(* Logix 5000 project; controller RSL5k_18_Template_noLib Emulate 5570 rev 32.11; software revision 32.02; part 5 of 16 *)
(* tags used below, declared in another part *)
   Inp_Hand : BOOL;   // 1=Acquire Hand (typ. hardwired local), 0=Release Hand
   Inp_Ovrd : BOOL;   // 1=Acquire Override (higher priority program logic), 0=Release Override
   Inp_ExtInh : BOOL;   // 1=Inhibit External Acquisition, 0=Allow External Acquisition
   Cfg_HasOper : BOOL;   // 1=Operator (unlocked) exists, can be selected
   Cfg_HasOperLocked : BOOL;   // 1=Operator Locked exists, can be selected
   Cfg_HasProg : BOOL;   // 1=Program (unlocked) exists, can be selected
   Cfg_HasProgLocked : BOOL;   // 1=Program Locked exists, can be selected
   Cfg_HasExt : BOOL;   // 1=External exists, can be selected
   Cfg_HasMaint : BOOL;   // 1=Maintenance exists, can be selected
   Cfg_HasMOoS : BOOL;   // 1=Maintenance Out of Service exists, can be selected
   Cfg_OvrdOverLock : BOOL;   // 1=Override supersedes Prog/Oper Lock, 0=don't override Lock
   Cfg_ExtOverLock : BOOL;   // 1=External supersedes Prog/Oper Lock, 0=don't override Lock
   Cfg_ProgNormal : BOOL;   // Normal Source: 1=Program if no requests; 0=Operator if no requests
   Cfg_PCmdPriority : BOOL;   // Command Priority: 1=Program Cmds Win; 0=Operator Cmds Win
   Cfg_PCmdProgAsLevel : BOOL;   // 1=PCmd_Prog used as a Level (1=Prog, 0=Oper)
   Cfg_PCmdLockAsLevel : BOOL;   // 1=PCmd_Lock used as a Level (1=Lock, 0=Unlock)
   Cfg_ExtAcqAsLevel : BOOL;   // 1=XCmd_Acq used as Level (1=Acq, 0=Rel)
   PCmd_Prog : BOOL;   // Program Command to select Program (Oper to Prog)
   PCmd_Lock : BOOL;   // Program Command to Lock Program (disallow Operator)
   MCmd_Acq : BOOL;   // Maintenance Command to Acquire (Oper/Prog/Ovrd to Maint)
   XCmd_Acq : BOOL;   // External Command to Acquire
   XCmd_Rel : BOOL;   // External Command to Release
   OCmd_Lock : BOOL;   // Operator Command to Lock Operator (disallow Program)
   Sts_eSrc : INT;   // Selection enum: .8=Ext, .7=OoS, .6=Oper, .5=Prog, .4=Ovrd, .3=Maint, .2=Hand, .1=Norm, .0=Lock
   Sts_bSrc : INT;   // Active Selection bitmap (for HMI totem pole)
   Sts_Hand : BOOL;   // 1=Hand is selected (supersedes OoS, Maint, Ovrd, Ext, Prog, Oper)
   Sts_OoS : BOOL;   // 1=Out of Service is selected (supersedes Maint, Ovrd, Ext, Prog, Oper)
   Sts_Maint : BOOL;   // 1=Maintenance is selected (supersedes Ovrd, Ext, Prog, Oper)
   Sts_Ovrd : BOOL;   // 1=Override is selected (supersedes Ext, Prog, Oper)
   Sts_Ext : BOOL;   // 1=External is selected (supersedes Prog, Oper)
   Sts_Prog : BOOL;   // 1=Program is selected
   Sts_ProgLocked : BOOL;   // 1=Program is selected and Locked
   Sts_Oper : BOOL;   // 1=Operator is selected
   Sts_OperLocked : BOOL;   // 1=Operator is selected and Locked
   Sts_ProgOperSel : BOOL;   // Prog/Oper selection (latch) state, 1=Program, 0=Operator
   Sts_ProgOperLock : BOOL;   // Prog/Oper lock (latch) state, 1=Locked, 0=Unlocked
   Sts_Normal : BOOL;   // 1=Selection equals the Normal (Prog or Oper)
   Sts_ProgReqInh : BOOL;   // 1=Program request inhibited, cannot Get to Program from Current State
   Sts_ExtReqInh : BOOL;   // 1=External request inhibited
   Sts_MAcqRcvd : BOOL;   // 1=Maintenance Acquire command received this scan
   MRdy_OoS : BOOL;   // 1=Ready for MCmd_OoS (enables HMI button)
   MRdy_IS : BOOL;   // 1=Ready for MCmd_IS (enables HMI button)
   MRdy_Acq : BOOL;   // 1=Ready for MCmd_Acq (enables HMI button)
   MRdy_Rel : BOOL;   // 1=Ready for MCmd_Rel (enables HMI button)
   XRdy_Acq : BOOL;   // 1=Ready for XCmd_Acq (enables HMI button)
   XRdy_Rel : BOOL;   // 1=Ready for XCmd_Rel (enables HMI button)
   ORdy_Oper : BOOL;   // 1=Ready for OCmd_Oper (enables HMI button)
   ORdy_Prog : BOOL;   // 1=Ready for OCmd_Prog (enables HMI button)
   ORdy_Lock : BOOL;   // 1=Ready for OCmd_Lock (enables HMI button)
   ORdy_Unlock : BOOL;   // 1=Ready for OCmd_Unlock (enables HMI button)
   ORdy_Normal : BOOL;   // 1=Ready for OCmd_Normal (enables HMI button)
   P_CmdSrc : BOOL;   // Unique Parameter Name for auto - discovery
   Wrk_ProgOperSel : BOOL;   // Internal Program (1) / Operator (0) selection result
   Wrk_ProgOperLock : BOOL;   // Internal Prog/Oper Lock (1) / Unlock (0) selection result
   Wrk_Prog : BOOL;   // Internal Program (1) / Operator (0) selection progress
   Wrk_MOoS : BOOL;   // Internal Maintenance Out of Service (1) / In Service (0) latch
   Wrk_Maint : BOOL;   // Internal Maintenance Acquire (1) / Release (0) latch
   Wrk_Lock : BOOL;   // Internal Prog/Oper Lock (1) / Unlock (0) selection progress
   Wrk_Init : BOOL;   // 1=Initialized, 0=Initialization is required (e.g., powerup)
   Wrk_Ext : BOOL;   // Internal latch of External selection (1=Ext acquired)
(* P_CmdSrc, continued *)

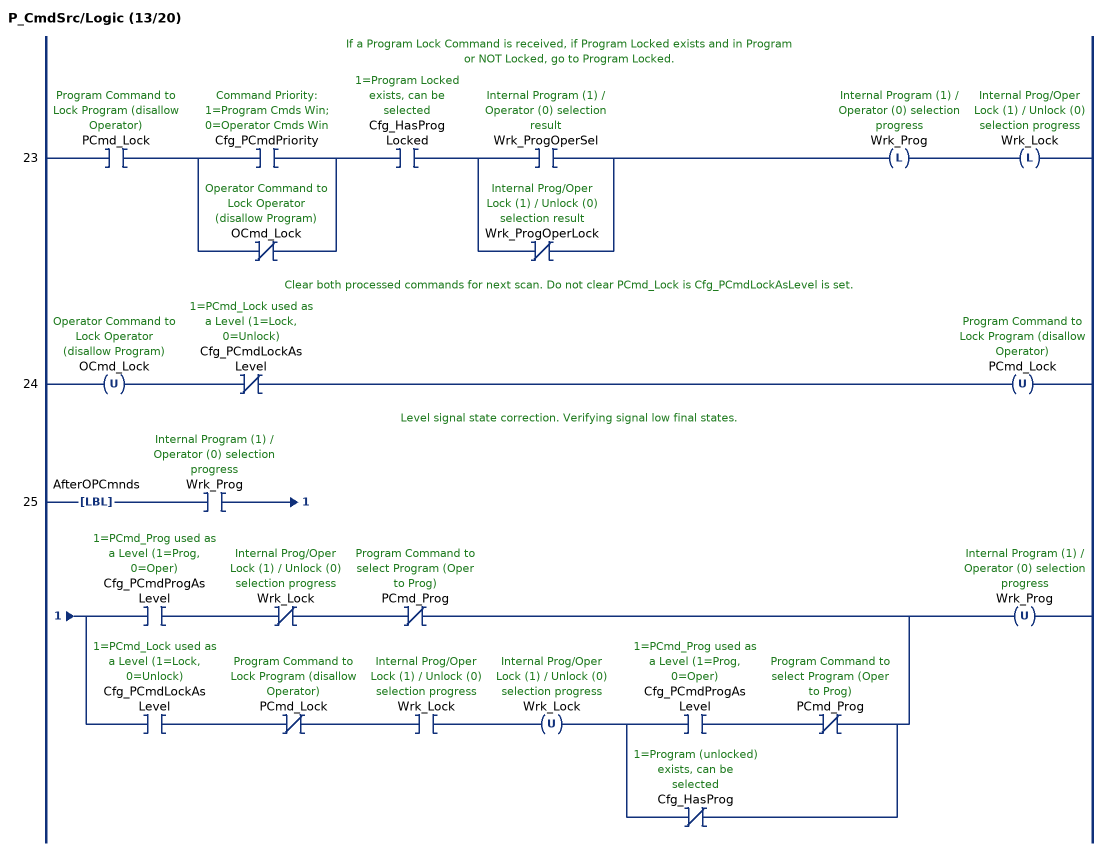
   // If a Program Lock Command is received, if Program Locked exists and in Program
   // or NOT Locked, go to Program Locked.
   23: XIC(PCmd_Lock)[XIC(Cfg_PCmdPriority) ,XIO(OCmd_Lock) ]XIC(Cfg_HasProgLocked)[XIC(Wrk_ProgOperSel) ,XIO(Wrk_ProgOperLock) ]OTL(Wrk_Prog)OTL(Wrk_Lock);
   // Clear both processed commands for next scan. Do not clear PCmd_Lock is Cfg_PCmdLockAsLevel is set.
   24: OTU(OCmd_Lock)XIO(Cfg_PCmdLockAsLevel)OTU(PCmd_Lock);
   // Level signal state correction. Verifying signal low final states.
   25: LBL(AfterOPCmnds)XIC(Wrk_Prog)[XIC(Cfg_PCmdProgAsLevel) XIO(Wrk_Lock) XIO(PCmd_Prog) ,XIC(Cfg_PCmdLockAsLevel) XIO(PCmd_Lock) XIC(Wrk_Lock) OTU(Wrk_Lock) [XIC(Cfg_PCmdProgAsLevel) XIO(PCmd_Prog) ,XIO(Cfg_HasProg) ] ]OTU(Wrk_Prog);
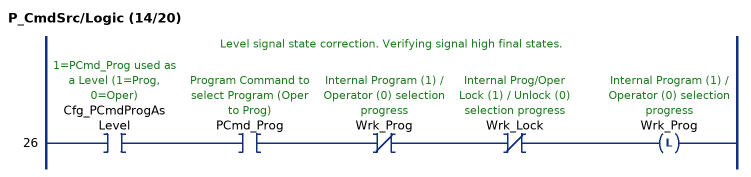
   // Level signal state correction. Verifying signal high final states.
   26: XIC(Cfg_PCmdProgAsLevel)XIC(PCmd_Prog)XIO(Wrk_Prog)XIO(Wrk_Lock)OTL(Wrk_Prog);
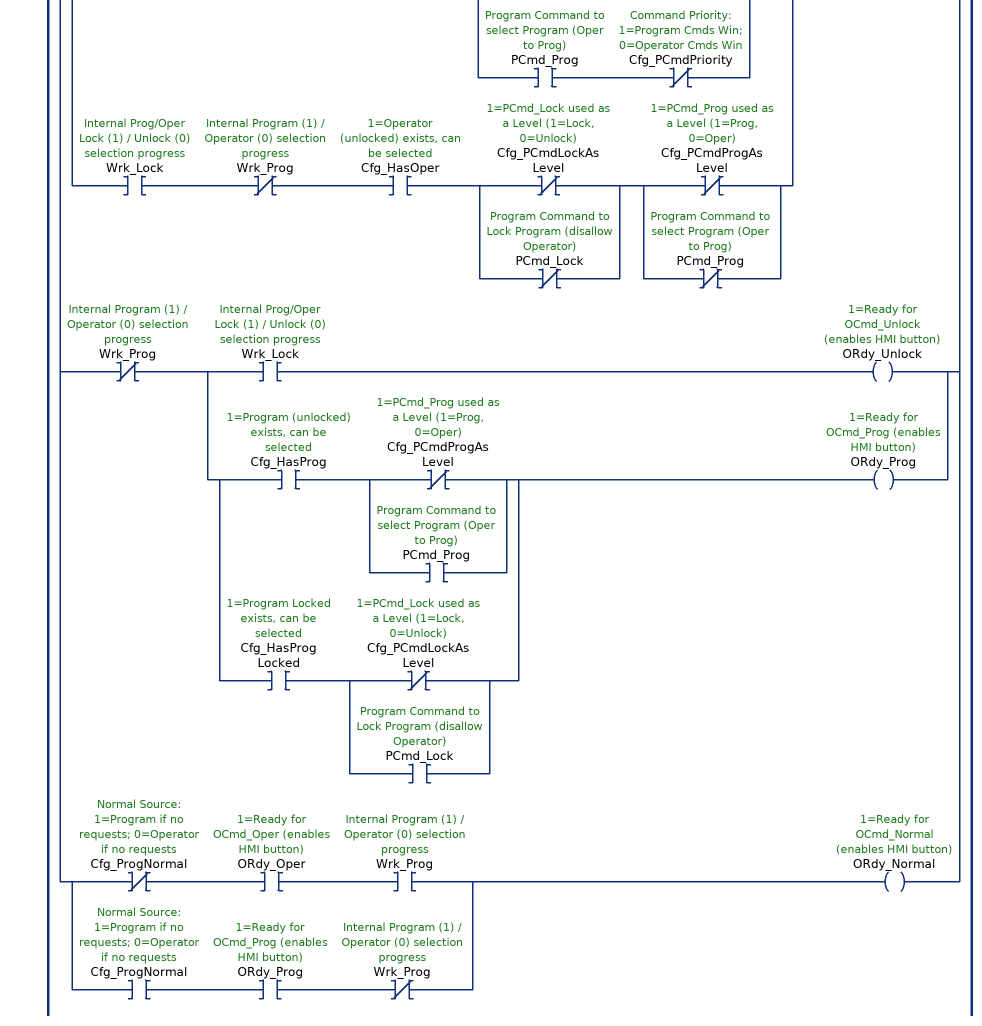
   // ============================================================
   // MAINTENANCE AND OPERATOR COMMAND READIES
   // ============================================================
   // This rung generates the "ORdy_" and "MRdy_" bits that signify to the
   // HMI that the corresponding command should "do" something
   // and the command button should be enabled on the display.
   // NOTE ON MAINTENANCE ACQUIRE: Ready for MCmd_Acq if Maintenance
   // is allowed and the internal Maintenance latch is NOT set.  However,
   // we need to display Ready even if latch IS set so that Sts_MAcqRcvd
   // can blink to reset an external Maintenance expiration timer!!!
   // #####  V4.10.00  2019-03-08:  Added XRdy_Acq, XRdy_Rel so External Acq/Rel can be used on HMI .  #####
   27: [XIC(Cfg_HasMaint) [OTE(MRdy_Acq) ,XIC(Wrk_Maint) OTE(MRdy_Rel) ] ,XIC(Cfg_HasMOoS) [XIC(Wrk_MOoS) OTE(MRdy_IS) ,XIO(Wrk_MOoS) OTE(MRdy_OoS) ] ,XIC(Cfg_HasExt) XIO(Cfg_ExtAcqAsLevel) [XIC(Wrk_Ext) OTE(XRdy_Rel) ,XIO(Wrk_Ext) XIO(Inp_ExtInh) OTE(XRdy_Acq) ] ,XIO(Wrk_Lock) XIC(Cfg_HasOperLocked) OTE(ORdy_Lock) ,[XIO(Wrk_Lock) XIC(Wrk_Prog) [XIC(Cfg_HasOper) XIO(Cfg_PCmdProgAsLevel) ,XIC(Cfg_HasOperLocked) [XIO(Cfg_PCmdProgAsLevel) ,XIC(PCmd_Prog) XIO(Cfg_PCmdPriority) ] ] ,XIC(Wrk_Lock) XIO(Wrk_Prog) XIC(Cfg_HasOper) [XIO(Cfg_PCmdLockAsLevel) ,XIO(PCmd_Lock) ] [XIO(Cfg_PCmdProgAsLevel) ,XIO(PCmd_Prog) ] ] OTE(ORdy_Oper) ,XIO(Wrk_Prog) [XIC(Wrk_Lock) OTE(ORdy_Unlock) ,[XIC(Cfg_HasProg) [XIO(Cfg_PCmdProgAsLevel) ,XIC(PCmd_Prog) ] ,XIC(Cfg_HasProgLocked) [XIO(Cfg_PCmdLockAsLevel) ,XIC(PCmd_Lock) ] ] OTE(ORdy_Prog) ] ,[XIO(Cfg_ProgNormal) XIC(ORdy_Oper) XIC(Wrk_Prog) ,XIC(Cfg_ProgNormal) XIC(ORdy_Prog) XIO(Wrk_Prog) ] OTE(ORdy_Normal) ];
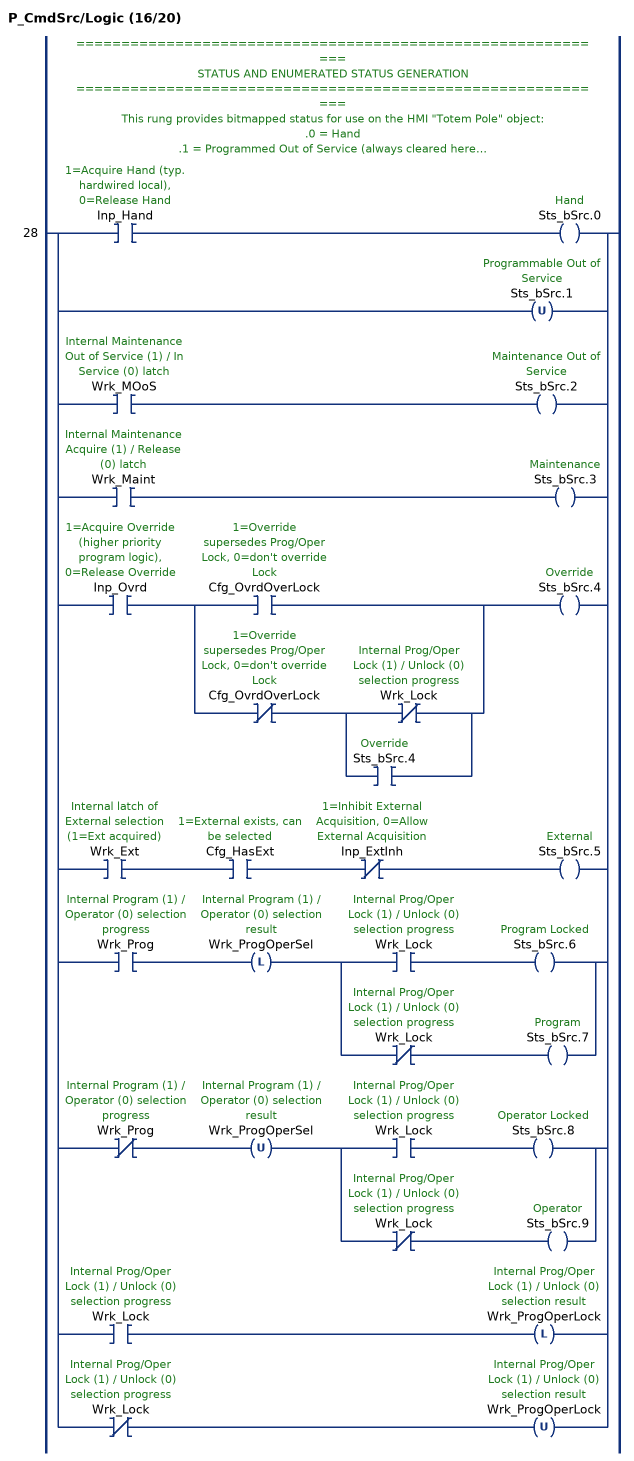
   // ============================================================
   // STATUS AND ENUMERATED STATUS GENERATION
   // ============================================================
   // This rung provides bitmapped status for use on the HMI "Totem Pole" object:
   // .0 = Hand
   // .1 = Programmed Out of Service (always cleared here)
   // .2 = Maintenance Out of Service
   // .3 = Maintenance
   // .4= Override
   // .5 = External
   // .6 = Program Locked
   // .7 = Program
   // .8 = Operator Locked
   // .9 = Operator
   // In addition, the final selections of the Program / Operator selection latch
   // and the Prog/Oper lock latch are captured for use next scan.
   // #####  V4.10.00  2019-03-08:  Added XCmd_Acq, XCmd_Rel, Cfg_ExtAcqAsLevel, removed Inp_Ext.  #####
   28: [XIC(Inp_Hand) OTE(Sts_bSrc.0) ,OTU(Sts_bSrc.1) ,XIC(Wrk_MOoS) OTE(Sts_bSrc.2) ,XIC(Wrk_Maint) OTE(Sts_bSrc.3) ,XIC(Inp_Ovrd) [XIC(Cfg_OvrdOverLock) ,XIO(Cfg_OvrdOverLock) [XIO(Wrk_Lock) ,XIC(Sts_bSrc.4) ] ] OTE(Sts_bSrc.4) ,XIC(Wrk_Ext) XIC(Cfg_HasExt) XIO(Inp_ExtInh) OTE(Sts_bSrc.5) ,XIC(Wrk_Prog) OTL(Wrk_ProgOperSel) [XIC(Wrk_Lock) OTE(Sts_bSrc.6) ,XIO(Wrk_Lock) OTE(Sts_bSrc.7) ] ,XIO(Wrk_Prog) OTU(Wrk_ProgOperSel) [XIC(Wrk_Lock) OTE(Sts_bSrc.8) ,XIO(Wrk_Lock) OTE(Sts_bSrc.9) ] ,XIC(Wrk_Lock) OTL(Wrk_ProgOperLock) ,XIO(Wrk_Lock) OTU(Wrk_ProgOperLock) ];
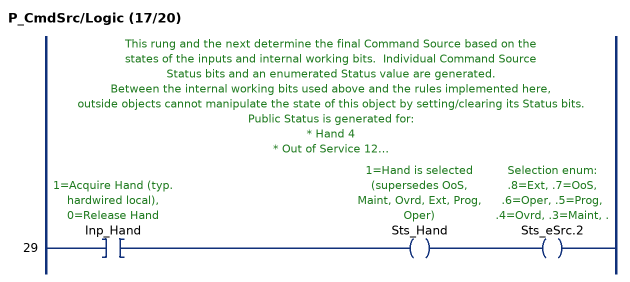
   // This rung and the next determine the final Command Source based on the
   // states of the inputs and internal working bits.  Individual Command Source
   // Status bits and an enumerated Status value are generated.
   // Between the internal working bits used above and the rules implemented here,
   // outside objects cannot manipulate the state of this object by setting/clearing its Status bits.
   // Public Status is generated for:
   // * Hand 4
   // * Out of Service 129
   // * Maintenance 8
   // * Override 16
   // * External 256
   // * Program 32
   // * Operator 64
   // * Program / Operator Lock status 33/65
   // * Command Source = Normal 34/66
   29: XIC(Inp_Hand)OTE(Sts_Hand)OTE(Sts_eSrc.2);
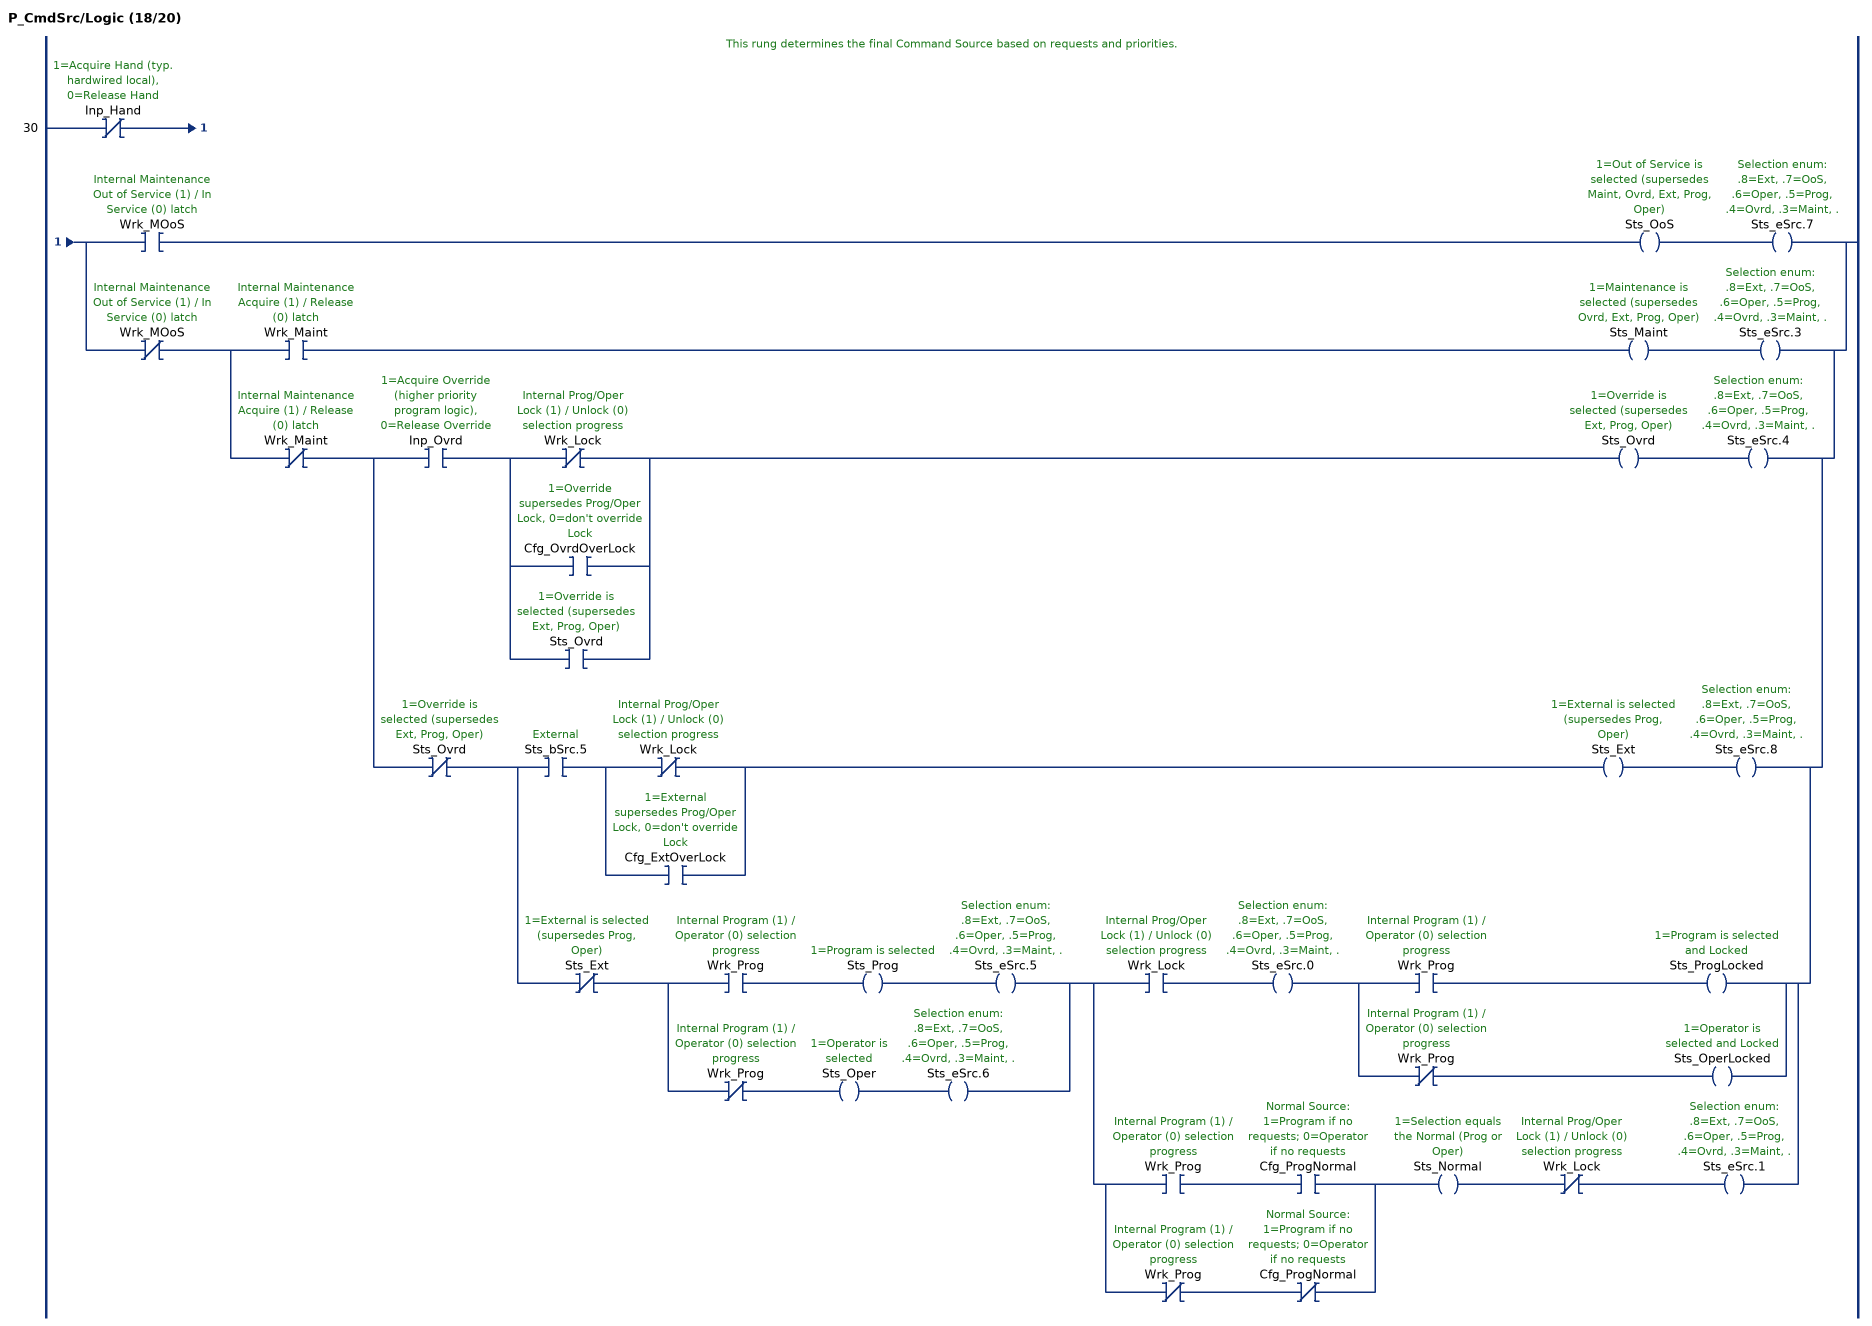
   // This rung determines the final Command Source based on requests and priorities.
   30: XIO(Inp_Hand)[XIC(Wrk_MOoS) OTE(Sts_OoS) OTE(Sts_eSrc.7) ,XIO(Wrk_MOoS) [XIC(Wrk_Maint) OTE(Sts_Maint) OTE(Sts_eSrc.3) ,XIO(Wrk_Maint) [XIC(Inp_Ovrd) [XIO(Wrk_Lock) ,XIC(Cfg_OvrdOverLock) ,XIC(Sts_Ovrd) ] OTE(Sts_Ovrd) OTE(Sts_eSrc.4) ,XIO(Sts_Ovrd) [XIC(Sts_bSrc.5) [XIO(Wrk_Lock) ,XIC(Cfg_ExtOverLock) ] OTE(Sts_Ext) OTE(Sts_eSrc.8) ,XIO(Sts_Ext) [XIC(Wrk_Prog) OTE(Sts_Prog) OTE(Sts_eSrc.5) ,XIO(Wrk_Prog) OTE(Sts_Oper) OTE(Sts_eSrc.6) ] [XIC(Wrk_Lock) OTE(Sts_eSrc.0) [XIC(Wrk_Prog) OTE(Sts_ProgLocked) ,XIO(Wrk_Prog) OTE(Sts_OperLocked) ] ,[XIC(Wrk_Prog) XIC(Cfg_ProgNormal) ,XIO(Wrk_Prog) XIO(Cfg_ProgNormal) ] OTE(Sts_Normal) XIO(Wrk_Lock) OTE(Sts_eSrc.1) ] ] ] ] ];
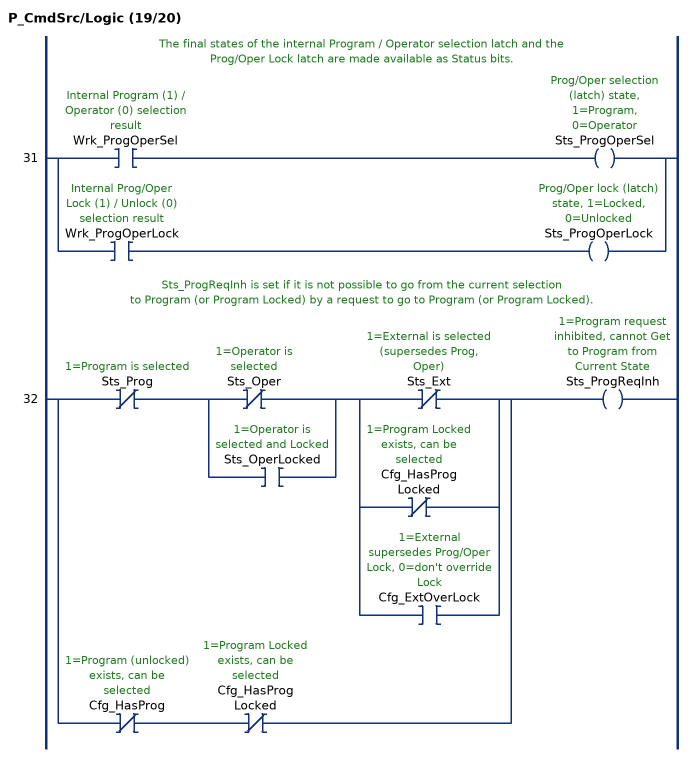
   // The final states of the internal Program / Operator selection latch and the
   // Prog/Oper Lock latch are made available as Status bits.
   31: [XIC(Wrk_ProgOperSel) OTE(Sts_ProgOperSel) ,XIC(Wrk_ProgOperLock) OTE(Sts_ProgOperLock) ];
   // Sts_ProgReqInh is set if it is not possible to go from the current selection
   // to Program (or Program Locked) by a request to go to Program (or Program Locked).
   32: [XIO(Sts_Prog) [XIO(Sts_Oper) ,XIC(Sts_OperLocked) ] [XIO(Sts_Ext) ,XIO(Cfg_HasProgLocked) ,XIC(Cfg_ExtOverLock) ] ,XIO(Cfg_HasProg) XIO(Cfg_HasProgLocked) ]OTE(Sts_ProgReqInh);
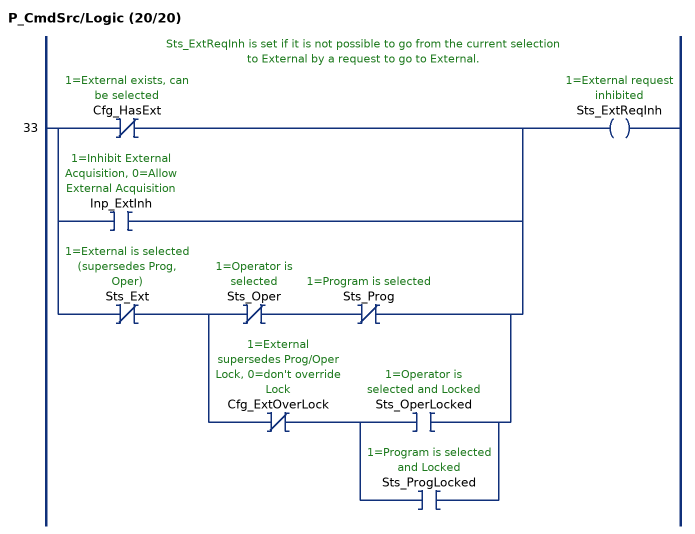
   // Sts_ExtReqInh is set if it is not possible to go from the current selection
   // to External by a request to go to External.
   33: [XIO(Cfg_HasExt) ,XIC(Inp_ExtInh) ,XIO(Sts_Ext) [XIO(Sts_Oper) XIO(Sts_Prog) ,XIO(Cfg_ExtOverLock) [XIC(Sts_OperLocked) ,XIC(Sts_ProgLocked) ] ] ]OTE(Sts_ExtReqInh);
END_ROUTINE

ROUTINE Prescan   (* ladder *)
// Sets internal state and enumerated / bit status to "not initialized".
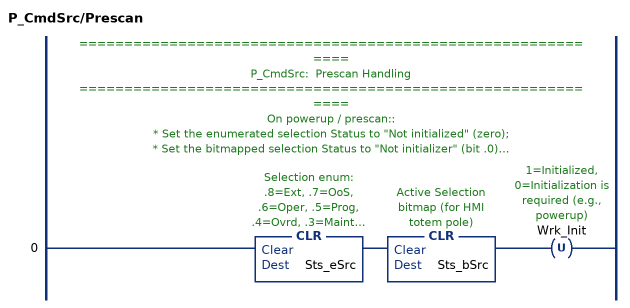
   // ============================================================
   // P_CmdSrc:  Prescan Handling
   // ============================================================
   // On powerup / prescan::
   // * Set the enumerated selection Status to "Not initialized" (zero);
   // * Set the bitmapped selection Status to "Not initializer" (bit .0);
   // * Flag the instruction to execute the initialization rungs when run.
   0: CLR(Sts_eSrc)CLR(Sts_bSrc)OTU(Wrk_Init);
END_ROUTINE
END_ADD_ON_INSTRUCTION

ADD_ON_INSTRUCTION P_Gate   (* revision 4.10 .00 Release, vendor Rockwell Automation, ExecutePrescan, ExecuteEnableInFalse *)
// Condition Gate/Delay
// Revision note:
// See Instruction Help for a summary of changes, and see 4.10 Release Notes for details.
// Help:
// Copyright © Rockwell Automation, Inc.  All Rights Reserved.
// This Instruction provides a "gate" for a discrete Input signal and
// provides on-delay and off-delay timing for the gated signal.
// When the Gate input is true, the instruction Input is passed through
// to the Output, with on-delay and off-delay timing applied.
// When the Gate input is false, the Output is kept off
// (note: off-delay still applies!)
// This instruction is usually used between a comparison
// (analog threshold with deadband or discrete logic)
// and a P_Alarm instance, but may be used as a
// gated on-delay/off-delay timer generally.
// When EnableIn  is FALSE (e.g., on a false LD rung), the Input "Inp"
// is inverted.  Note that the Gate input (Inp_Gate) is NOT inverted!!!
// SUMMARY OF CHANGES FROM PREVIOUS VERSION (4.00.00)
// See 4.10 Release Notes for details.
// * Unmodified, up-rev only for Library 4.10.00
// SUMMARY OF CHANGES FROM PREVIOUS VERSION (3.5-01)
// See 4.00 Release Notes for details.
// * Changed Inf_ items to HMI_ (e.g., HMI_Lib, HMI_Type).
// * Changed delay time configuration items to REAL seconds
VAR_INPUT
   Inp : BOOL; {visible}   // Input Condition: e.g., result of comparison
   Inp_Gate : BOOL := 1; {visible}   // Gate Input: 1=enable On Delay / Off Delay after Gate Delay, 0=disable
   Cfg_GateDly : REAL;   // Gate Delay (s): time after Gate Input true to enable On/Off Delay
   Cfg_OnDly : REAL;   // On Delay (s): If Gate Delay done, time Inp must be true to set Out true
   Cfg_OffDly : REAL;   // Off Delay (s): Time after Inp or Gate goes to 0 for Out to go to 0
END_VAR
VAR_OUTPUT
   Out : BOOL; {access Read Only, visible}   // Output after On Delay, Off Delay, enabled by Gate
   Sts_Gate : BOOL; {access Read Only, visible}   // 1=Gate Delay done, Output is enabled
   Sts_Err : BOOL; {access Read Only, visible}   // 1=Error in Config (see detail Err_ bits for reason), display icon
   Err_Timer : BOOL; {access Read Only}   // 1=Error in Config: On Delay, Off Delay, Gate Delay Time Invalid (use 0 to 2147483 s)
   P_Gate : BOOL;   // Unique Parameter Name for auto - discovery
END_VAR
VAR
   Wrk_OffDlyT : TIMER; {access Read Only}   // Off Delay Timer
   Wrk_OnDlyT : TIMER; {access Read Only}   // On Delay Timer
   Wrk_GateT : TIMER; {access Read Only}   // Gate Delay Timer
   Cfg_InpCond : STRING_20 := 'Input Condition';   // Displayed text of P_Gate's Input (Inp) Condition
   HMI_Lib : STRING_12 := 'RA-BAS'; {access Read Only}   // Display Library for Faceplate call-up
   HMI_Type : STRING_16 := 'P_Gate'; {access Read Only}   // Must contain AOI name, used for HMI and Information S/W
   Cfg_GateCond : STRING_20 := 'Gating Condition';   // Displayed text of P_Gate's Gating (Inp_Gate) Condition
   HMI_Tab : SINT;   // Tab to display (FTView ME)
END_VAR

ROUTINE EnableInFalse   (* ladder *)
// Same as main Logic routine, except Inp is inverted (for use in LD logic)  (Inp_Gate is NOT inverted!!!)
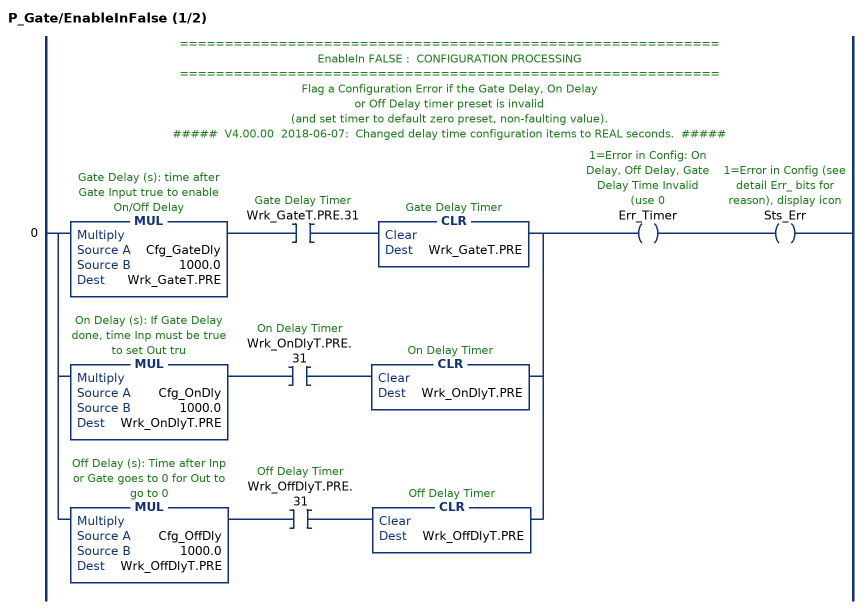
   // ============================================================
   // EnableIn FALSE :  CONFIGURATION PROCESSING
   // ============================================================
   // Flag a Configuration Error if the Gate Delay, On Delay
   // or Off Delay timer preset is invalid
   // (and set timer to default zero preset, non-faulting value).
   // #####  V4.00.00  2018-06-07:  Changed delay time configuration items to REAL seconds.  #####
   0: [MUL(Cfg_GateDly,1000.0,Wrk_GateT.PRE) XIC(Wrk_GateT.PRE.31) CLR(Wrk_GateT.PRE) ,MUL(Cfg_OnDly,1000.0,Wrk_OnDlyT.PRE) XIC(Wrk_OnDlyT.PRE.31) CLR(Wrk_OnDlyT.PRE) ,MUL(Cfg_OffDly,1000.0,Wrk_OffDlyT.PRE) XIC(Wrk_OffDlyT.PRE.31) CLR(Wrk_OffDlyT.PRE) ]OTE(Err_Timer)OTE(Sts_Err);
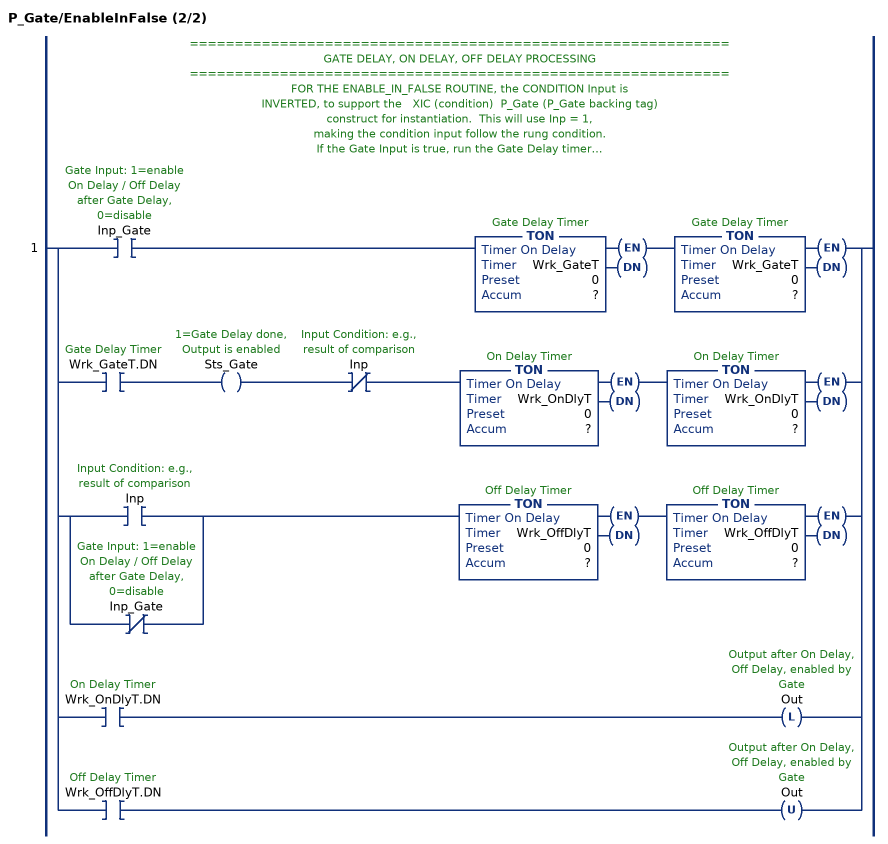
   // ============================================================
   // GATE DELAY, ON DELAY, OFF DELAY PROCESSING
   // ============================================================
   // FOR THE ENABLE_IN_FALSE ROUTINE, the CONDITION Input is
   // INVERTED, to support the   XIC (condition)  P_Gate (P_Gate backing tag)
   // construct for instantiation.  This will use Inp = 1,
   // making the condition input follow the rung condition.
   // If the Gate Input is true, run the Gate Delay timer.
   // Once the Gate Delay is complete, enable the
   // On Delay and Off Delay that follow the INVERTED input.
   // Report the Gate Delay status and the final Output status (after all delays).
   // @@@@@  NOTE: Doubled TONs are used to ensure that  @@@@@
   // @@@@@  .DN bit transitions on same scan if Preset = 0 !  @@@@@
   1: [XIC(Inp_Gate) TON(Wrk_GateT,?,?) TON(Wrk_GateT,?,?) ,XIC(Wrk_GateT.DN) OTE(Sts_Gate) XIO(Inp) TON(Wrk_OnDlyT,?,?) TON(Wrk_OnDlyT,?,?) ,[XIC(Inp) ,XIO(Inp_Gate) ] TON(Wrk_OffDlyT,?,?) TON(Wrk_OffDlyT,?,?) ,XIC(Wrk_OnDlyT.DN) OTL(Out) ,XIC(Wrk_OffDlyT.DN) OTU(Out) ];
END_ROUTINE

ROUTINE Logic   (* ladder *)
// Gate the input and apply on-delay and off-delay timing
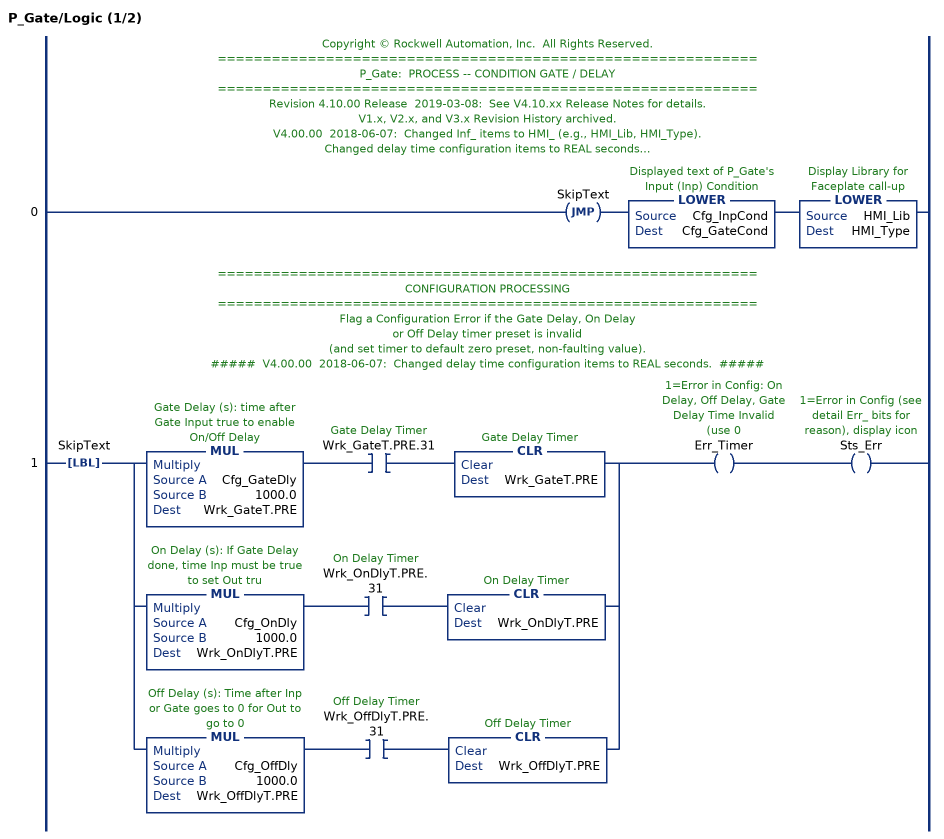
   // Copyright © Rockwell Automation, Inc.  All Rights Reserved.
   // ============================================================
   // P_Gate:  PROCESS -- CONDITION GATE / DELAY
   // ============================================================
   // Revision 4.10.00 Release  2019-03-08:  See V4.10.xx Release Notes for details.
   // V1.x, V2.x, and V3.x Revision History archived.
   // V4.00.00  2018-06-07:  Changed Inf_ items to HMI_ (e.g., HMI_Lib, HMI_Type).
   // Changed delay time configuration items to REAL seconds.
   // V4.10.00  2019-03-08:  Unmodified, up-rev only for Library 4.10.00
   // ============================================================
   // This Instruction provides a "gate" for a discrete Input signal and
   // provides on-delay and off-delay timing for the gated signal.
   // When the Gate input is true, the instruction Input is passed through
   // to the Output, with on-delay and off-delay timing applied.
   // When the Gate input is false, the Output is kept off
   // (note: off-delay still applies!)
   // This instruction is usually used between a comparison
   // (analog threshold with deadband or discrete logic)
   // and a P_Alarm instance, but may be used as a
   // gated on-delay/off-delay timer generally.
   // When EnableIn  is FALSE (e.g., on a false LD rung),
   // the Input "Inp" is inverted.  Note that the Gate
   // input (Inp_Gate) is NOT inverted!!!
   // ============================================================
   // SHOW LOCAL STRINGS
   // ============================================================
   // The STRINGs containing the text associated with each instance of this
   // instruction cannot be Input or Output Parameters, because STRINGs are not
   //  'atomic' types. (Inputs and Outputs must be SINT, INT, DINT, REAL, or BOOL.)
   // In order to make it easier to find and configure these STRINGs, this rung
   // was added.  THE JMP (and the LBL on the following rung)
   // MUST NOT BE REMOVED!!!
   // To view the STRINGs, go to the instruction instance (in LD or FBD), RIGHT-click
   // to bring up the context menu and select "Open Instruction Logic".
   // This rung will appear with the STRING values for the selected instance.
   // You may double-click the STRING values here to modify them as well.
   0: JMP(SkipText)LOWER(Cfg_InpCond,Cfg_GateCond)LOWER(HMI_Lib,HMI_Type);
   // ============================================================
   // CONFIGURATION PROCESSING
   // ============================================================
   // Flag a Configuration Error if the Gate Delay, On Delay
   // or Off Delay timer preset is invalid
   // (and set timer to default zero preset, non-faulting value).
   // #####  V4.00.00  2018-06-07:  Changed delay time configuration items to REAL seconds.  #####
   1: LBL(SkipText)[MUL(Cfg_GateDly,1000.0,Wrk_GateT.PRE) XIC(Wrk_GateT.PRE.31) CLR(Wrk_GateT.PRE) ,MUL(Cfg_OnDly,1000.0,Wrk_OnDlyT.PRE) XIC(Wrk_OnDlyT.PRE.31) CLR(Wrk_OnDlyT.PRE) ,MUL(Cfg_OffDly,1000.0,Wrk_OffDlyT.PRE) XIC(Wrk_OffDlyT.PRE.31) CLR(Wrk_OffDlyT.PRE) ]OTE(Err_Timer)OTE(Sts_Err);
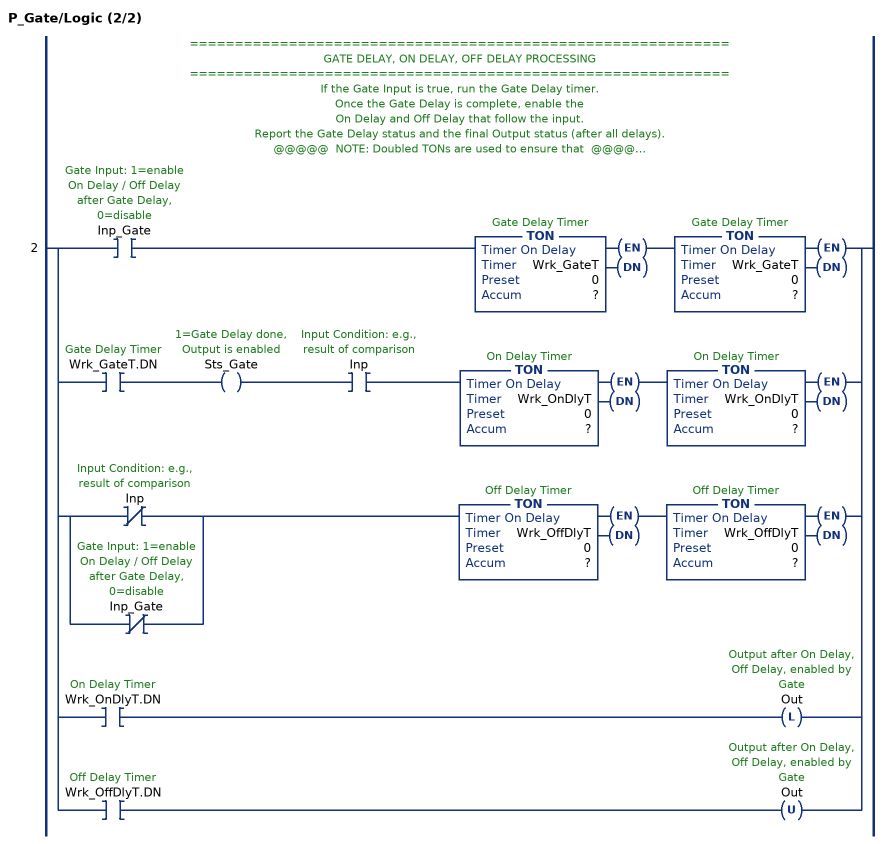
   // ============================================================
   // GATE DELAY, ON DELAY, OFF DELAY PROCESSING
   // ============================================================
   // If the Gate Input is true, run the Gate Delay timer.
   // Once the Gate Delay is complete, enable the
   // On Delay and Off Delay that follow the input.
   // Report the Gate Delay status and the final Output status (after all delays).
   // @@@@@  NOTE: Doubled TONs are used to ensure that  @@@@@
   // @@@@@  .DN bit transitions on same scan if Preset = 0 !  @@@@@
   2: [XIC(Inp_Gate) TON(Wrk_GateT,?,?) TON(Wrk_GateT,?,?) ,XIC(Wrk_GateT.DN) OTE(Sts_Gate) XIC(Inp) TON(Wrk_OnDlyT,?,?) TON(Wrk_OnDlyT,?,?) ,[XIO(Inp) ,XIO(Inp_Gate) ] TON(Wrk_OffDlyT,?,?) TON(Wrk_OffDlyT,?,?) ,XIC(Wrk_OnDlyT.DN) OTL(Out) ,XIC(Wrk_OffDlyT.DN) OTU(Out) ];
END_ROUTINE

ROUTINE Prescan   (* ladder *)
// Set the Gate Input to 1 (default value) on prescan
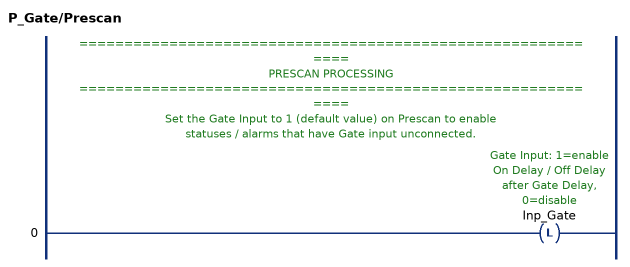
   // ============================================================
   // PRESCAN PROCESSING
   // ============================================================
   // Set the Gate Input to 1 (default value) on Prescan to enable
   // statuses / alarms that have Gate input unconnected.
   0: OTL(Inp_Gate);
END_ROUTINE
END_ADD_ON_INSTRUCTION

ADD_ON_INSTRUCTION P_Intlk   (* revision 4.10 .01 Release, vendor Rockwell Automation, ExecutePrescan, ExecuteEnableInFalse *)
// Interlocks
// Revision note:
// See Instruction Help for a summary of changes, and see 4.10 Release Notes for details.
// Help:
// Copyright © Rockwell Automation, Inc.  All Rights Reserved.
// This Instruction monitors up to 16 Interlock conditions.  It provides these features:
// *  The "OK" state of each Interlock Input is configurable.  By default,
//     each Input is 1 to trip, 0 when OK to run.
// *  Interlocks may be configured as Latched.  Latched Interlocks
//     require a Reset Command to clear.  The latching function can be
//     inhibited via a Latch Defeat input, for example, to avoid latching
//     Interlocks for a stopped motor.
// *  Interlocks may be configured as Bypassable; Non-Bypassable
//     Interlocks are reported separately so the destination object can
//     decide whether to bypass (ignore) bypassable interlocks, such
//     as in Maintenance Mode.
// *  First-Out reporting indicates the first condition that caused the
//     running equipment to be tripped.
// *  For each Interlock condition, a Tag may be defined for navigation.
//     Clicking the Interlock description will call up the associated Tag's
//     Faceplate.
// SUMMARY OF CHANGES FROM PREVIOUS VERSION (4.10.00)
// See 4.10 Release Notes for details.
// * Modified conditions for clearing first-out status and text.
// SUMMARY OF CHANGES FROM PREVIOUS VERSION (4.00.00)
// See 4.10 Release Notes for details.
// * Changed type of Val_FirstOutTxt to STRING_Cond.
// * Corrected Scan Mode selection to execute Prescan logic.
// * Added Cfg_HasMoreObj.
// SUMMARY OF CHANGES FROM PREVIOUS VERSION (3.5-05)
// See 4.00 Release Notes for details.
// * Changed Inf_ items to HMI_, and added Cfg_Area for security.
// * Added Val_FirstOutTxt string (Local, read-only) for use in
//    IntlkTrip alarm message  (ref: KnowledgeBase answer ID 672568).
// * Deleted Cfg_PCmdClear; all Program Commands are now self-clearing.
// * All OCmds/MCmds and ORdys/MRdys are now Local Tags.
// * Added Sts_RdyReset for use by external objects.
VAR_INPUT
   Inp_Intlk00 : ALIAS FOR Wrk_Inp.0; {visible}   // Interlock Cond. 00, Stop if not in configured OK state
   Inp_Intlk01 : ALIAS FOR Wrk_Inp.1; {visible}   // Interlock Cond. 01, Stop if not in configured OK state
   Inp_Intlk02 : ALIAS FOR Wrk_Inp.2; {visible}   // Interlock Cond. 02, Stop if not in configured OK state
   Inp_Intlk03 : ALIAS FOR Wrk_Inp.3; {visible}   // Interlock Cond. 03, Stop if not in configured OK state
   Inp_Intlk04 : ALIAS FOR Wrk_Inp.4; {visible}   // Interlock Cond. 04, Stop if not in configured OK state
   Inp_Intlk05 : ALIAS FOR Wrk_Inp.5; {visible}   // Interlock Cond. 05, Stop if not in configured OK state
   Inp_Intlk06 : ALIAS FOR Wrk_Inp.6; {visible}   // Interlock Cond. 06, Stop if not in configured OK state
   Inp_Intlk07 : ALIAS FOR Wrk_Inp.7; {visible}   // Interlock Cond. 07, Stop if not in configured OK state
   Inp_Intlk08 : ALIAS FOR Wrk_Inp.8;   // Interlock Cond. 08, Stop if not in configured OK state
   Inp_Intlk09 : ALIAS FOR Wrk_Inp.9;   // Interlock Cond. 09, Stop if not in configured OK state
   Inp_Intlk10 : ALIAS FOR Wrk_Inp.10;   // Interlock Cond. 10, Stop if not in configured OK state
   Inp_Intlk11 : ALIAS FOR Wrk_Inp.11;   // Interlock Cond. 11, Stop if not in configured OK state
   Inp_Intlk12 : ALIAS FOR Wrk_Inp.12;   // Interlock Cond. 12, Stop if not in configured OK state
   Inp_Intlk13 : ALIAS FOR Wrk_Inp.13;   // Interlock Cond. 13, Stop if not in configured OK state
   Inp_Intlk14 : ALIAS FOR Wrk_Inp.14;   // Interlock Cond. 14, Stop if not in configured OK state
   Inp_Intlk15 : ALIAS FOR Wrk_Inp.15;   // Interlock Cond. 15, Stop if not in configured OK state
   Inp_BypActive : BOOL; {visible}   // 1=Interlock Bypassing is currently active
   Inp_LatchDefeat : BOOL; {visible}   // Latch Defeat 1=Do not latch inputs even if configured for latching
   Inp_Reset : BOOL; {visible}   // 1=Reset Latched Interlocks and First-Out
   Cfg_OKState : INT;   // Bits indicate which state (0 or 1) of each input is OK to run
   Cfg_Latched : INT;   // Set bits indicate which conditions are latched (sealed in)
   Cfg_Bypassable : INT;   // Set bits indicate which conditions can be bypassed
   Cfg_HasNav : INT;   // Set bits indicate which Navigation buttons are enabled
   Cfg_HasMoreObj : BOOL;   // 1=Tells HMI an object with more info is available
   PCmd_Reset : BOOL;   // Program Command to Reset Latched Interlocks
END_VAR
VAR_OUTPUT
   Sts_IntlkOK : BOOL := 1; {access Read Only, visible}   // Overall Interlock Status (1=OK to run, 0=Stop)
   Sts_NBIntlkOK : BOOL := 1; {access Read Only, visible}   // Non-Bypassable Interlock Status (1=All NB Interlocks OK to run)
   Sts_BypActive : BOOL; {access Read Only}   // 1=Interlock Bypassing is Active (ignore bypassable interlocks)
   Sts_RdyReset : ALIAS FOR ORdy_Reset; {access Read Only}   // 1=A latched interlock (returned to OK) is ready to be reset
   Sts_Intlk : INT; {access Read Only, visible}   // Individual Interlock Status (1=Stop, 0=OK)
   Sts_FirstOut : INT; {access Read Only, visible}   // Interlock First Out Status (bit 1 is First Not-OK condition)
   P_Intlk : BOOL;   // Unique Parameter Name for auto - discovery
END_VAR
VAR
   Cfg_CondTxt : STRING_Cond[16] := ([0] := 'Enter Description #0');   // Short HMI description of Interlock Conditions
   Wrk_Inp : INT;   // Collection copy of Inp_IntlkXXs
   Wrk_NB : INT; {access None}   // Working register for Non-Bypassable Interlock ogic
   Wrk_Intlk : INT; {access None}   // Working register for Interlock logic
   Wrk_FirstOut : INT; {access None}   // Working register for First Out logic
   Wrk_Sts : INT; {access None}   // Working register for generating Interlock status
   Wrk_PrevSts : INT; {access None}   // Interlock Status previous scan
   Wrk_LatchEnable : BOOL := 1; {access None}   // 1=Latch interlock if configured to latch, 0=don't latch
   HMI_Tab : SINT;   // Tab to display (FTView ME)
   Wrk_InpInv : INT; {access None}   // Input states after inversion based on Cfg_OKState
   HMI_Type : STRING_16 := 'P_Intlk'; {access Read Only}   // Type identifier for HMI navigation
   Cfg_Label : STRING_20 := 'Interlocks';   // Label for graphic symbol displayed on HMI
   Cfg_Tag : STRING_20 := 'P_Intlk';   // Tagname for display on HMI
   Cfg_Desc : STRING_40 := 'Interlocks with First Out';   // Description for display on HMI
   Cfg_NavTag : STRING_NavTag[16];   // Tagnames for destinations of Navigation buttons
   HMI_Lib : STRING_12 := 'RA-BAS'; {access Read Only}   // Display Library for Faceplate call-up
   MSet_Bypass : INT;   // Individual condition Maintenance Bypass toggles
   Cfg_Area : STRING_Area := 'area01';   // Process Area for security
   Val_FirstOutTxt : STRING_Cond; {access Read Only}   // Text Description of First-Out Condition
   Wrk_NonIntlkStop : BOOL; {access None}   // One-Shot store: Stop OTHER than Interlock Stop occurred.
   Wrk_SetFirstOut : BOOL; {access None}   // One-Shot store: First Out update triggered
   ORdy_Reset : BOOL; {access Read Only}   // 1=Ready for OCmd_Reset (enables HMI button)
   OCmd_Reset : BOOL;   // Operator Command to Reset Latched Interlocks
END_VAR

ROUTINE EnableInFalse   (* ladder *)
// Set summary "OK" Status bits to FALSE (0)
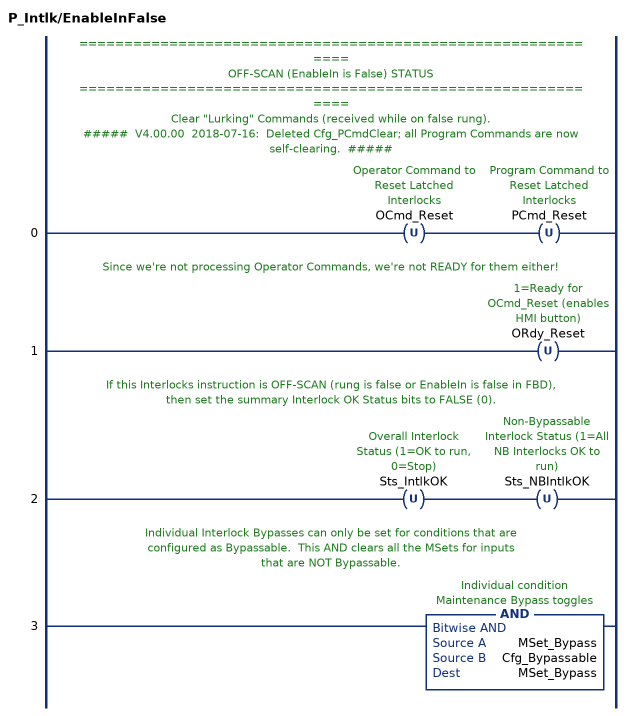
   // ============================================================
   // OFF-SCAN (EnableIn is False) STATUS
   // ============================================================
   //  Clear "Lurking" Commands (received while on false rung).
   // #####  V4.00.00  2018-07-16:  Deleted Cfg_PCmdClear; all Program Commands are now self-clearing.  #####
   0: OTU(OCmd_Reset)OTU(PCmd_Reset);
   // Since we're not processing Operator Commands, we're not READY for them either!
   1: OTU(ORdy_Reset);
   // If this Interlocks instruction is OFF-SCAN (rung is false or EnableIn is false in FBD),
   // then set the summary Interlock OK Status bits to FALSE (0).
   2: OTU(Sts_IntlkOK)OTU(Sts_NBIntlkOK);
   // Individual Interlock Bypasses can only be set for conditions that are
   // configured as Bypassable.  This AND clears all the MSets for inputs
   // that are NOT Bypassable.
   3: AND(MSet_Bypass,Cfg_Bypassable,MSet_Bypass);
END_ROUTINE

ROUTINE Logic   (* ladder *)
// Check Interlock Conditions
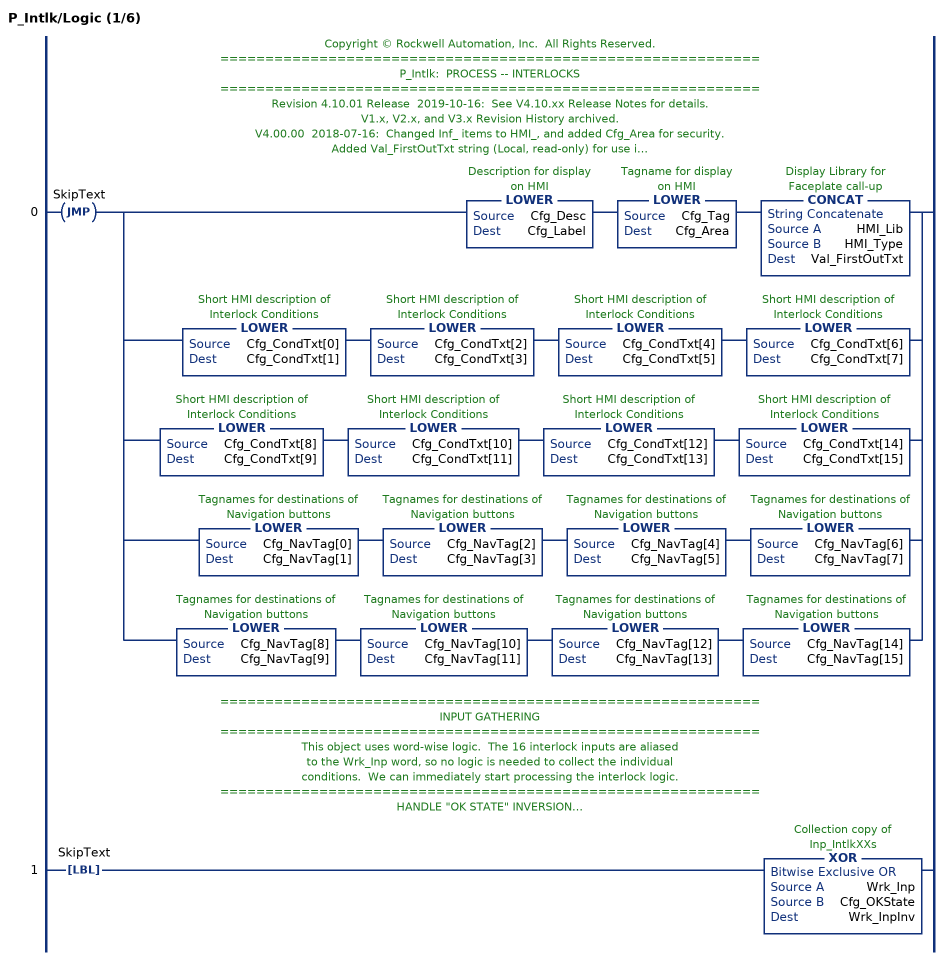
   // Copyright © Rockwell Automation, Inc.  All Rights Reserved.
   // ============================================================
   // P_Intlk:  PROCESS -- INTERLOCKS
   // ============================================================
   // Revision 4.10.01 Release  2019-10-16:  See V4.10.xx Release Notes for details.
   // V1.x, V2.x, and V3.x Revision History archived.
   // V4.00.00  2018-07-16:  Changed Inf_ items to HMI_, and added Cfg_Area for security.
   // Added Val_FirstOutTxt string (Local, read-only) for use in
   // IntlkTrip alarm message  (ref: KnowledgeBase answer ID 672568).
   // Deleted Cfg_PCmdClear; all Program Commands are now self-clearing.
   // All OCmds/MCmds and ORdys/MRdys are now Local Tags.
   // Added Sts_RdyReset for use by external objects.
   // V4.10.00  2019-03-08:  Changed type of Val_FirstOutTxt to STRING_Cond.
   // Corrected Scan Mode selection to execute Prescan logic. Added Cfg_HasMoreObj.\
   // V4.10.01  2019-10-16:  Modified conditions for clearing first-out status and text.
   // ============================================================
   // This Instruction monitors up to 16 Interlock conditions.  It provides these features:
   // *  The "OK" state of each Interlock Input is configurable.
   // By default, each Input is 1 to trip, 0 when OK to run.
   // *  Interlocks may be configured as Latched.  Latched Interlocks
   // require a Reset Command to clear.  The latching function can be inhibited
   // via a Latch Defeat input, for example, to avoid latching Interlocks for a stopped motor.
   // *  Interlocks may be configured as Bypassable.  Bypassable Interlocks are reported
   // separately; the destination object can use this information to bypass these
   // Interlocks in Maintenance Mode or upon command.
   // *  First-Out reporting indicates the first condition that
   // caused the running equipment to be tripped.
   // * For each Interlock condition, a Tag may be defined for navigation. Clicking
   // the Interlock description will call up the associated Tag's Faceplate.
   // ============================================================
   // SHOW LOCAL STRINGS
   // ============================================================
   // The STRINGs containing the text associated with each instance of this
   // instruction cannot be Input or Output Parameters, because STRINGs are not
   //  'atomic' types. (Inputs and Outputs must be SINT, INT, DINT, REAL, or BOOL.)
   // In order to make it easier to find and configure these STRINGs, this rung
   // was added.  THE JMP (and the LBL on the following rung)
   // MUST NOT BE REMOVED!!!
   // To view the STRINGs, go to the instruction instance (in LD or FBD), RIGHT-click
   // to bring up the context menu and select "Open Instruction Logic".
   // This rung will appear with the STRING values for the selected instance.
   // You may double-click the STRING values here to modify them as well.
   // #####  V4.00.00  2018-07-16:  Added string for Cfg_Area, Val_FirstOutTxt; renamed Inf_* to HMI_*.  #####
   0: JMP(SkipText)[LOWER(Cfg_Desc,Cfg_Label) LOWER(Cfg_Tag,Cfg_Area) CONCAT(HMI_Lib,HMI_Type,Val_FirstOutTxt) ,LOWER(Cfg_CondTxt[0],Cfg_CondTxt[1]) LOWER(Cfg_CondTxt[2],Cfg_CondTxt[3]) LOWER(Cfg_CondTxt[4],Cfg_CondTxt[5]) LOWER(Cfg_CondTxt[6],Cfg_CondTxt[7]) ,LOWER(Cfg_CondTxt[8],Cfg_CondTxt[9]) LOWER(Cfg_CondTxt[10],Cfg_CondTxt[11]) LOWER(Cfg_CondTxt[12],Cfg_CondTxt[13]) LOWER(Cfg_CondTxt[14],Cfg_CondTxt[15]) ,LOWER(Cfg_NavTag[0],Cfg_NavTag[1]) LOWER(Cfg_NavTag[2],Cfg_NavTag[3]) LOWER(Cfg_NavTag[4],Cfg_NavTag[5]) LOWER(Cfg_NavTag[6],Cfg_NavTag[7]) ,LOWER(Cfg_NavTag[8],Cfg_NavTag[9]) LOWER(Cfg_NavTag[10],Cfg_NavTag[11]) LOWER(Cfg_NavTag[12],Cfg_NavTag[13]) LOWER(Cfg_NavTag[14],Cfg_NavTag[15]) ];
   // ============================================================
   // INPUT GATHERING
   // ============================================================
   // This object uses word-wise logic.  The 16 interlock inputs are aliased
   // to the Wrk_Inp word, so no logic is needed to collect the individual
   // conditions.  We can immediately start processing the interlock logic.
   // ============================================================
   // HANDLE "OK STATE" INVERSIONS
   // ============================================================
   // This rung inverts the Input bits whose "OK State" is 1 (0 to Stop).
   // The resulting Wrk_Inp word is ZERO if all interlock inputs are "OK".
   1: LBL(SkipText)XOR(Wrk_Inp,Cfg_OKState,Wrk_InpInv);
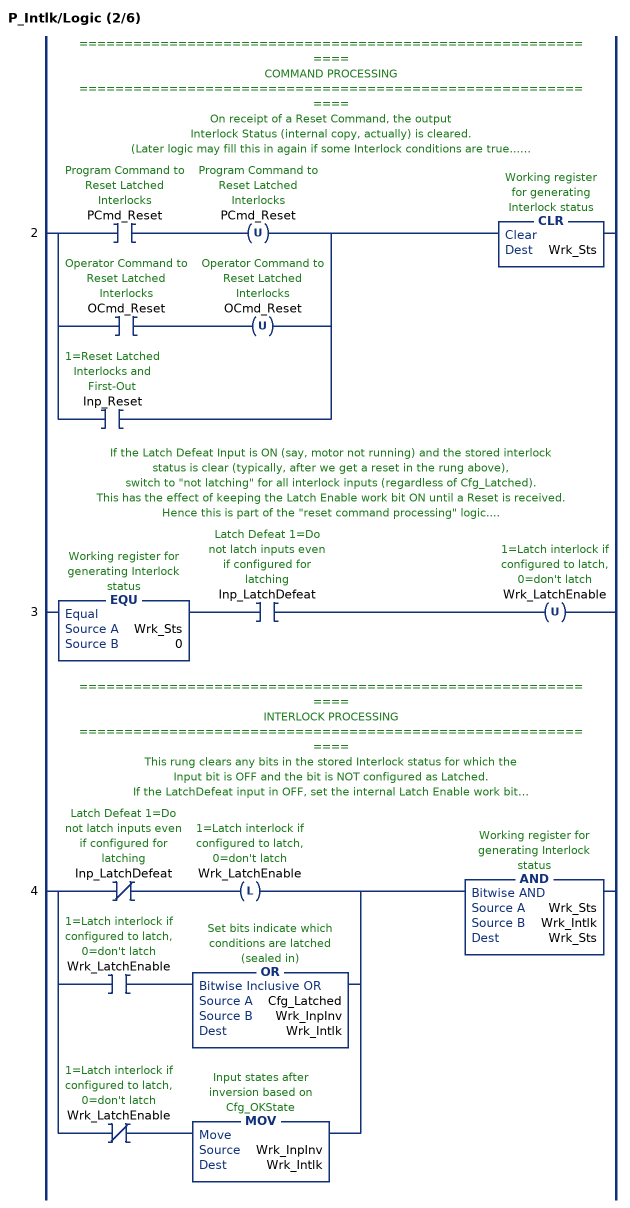
   // ============================================================
   // COMMAND PROCESSING
   // ============================================================
   // On receipt of a Reset Command, the output
   // Interlock Status (internal copy, actually) is cleared.
   // (Later logic may fill this in again if some Interlock conditions are true...)
   // NOTE:  This object is "Modeless" -- Operator and Program Commands
   // are accepted at any time.
   // #####  V4.00.00  2018-07-16:  Deleted Cfg_PCmdClear; all Program Commands are now self-clearing.  #####
   2: [XIC(PCmd_Reset) OTU(PCmd_Reset) ,XIC(OCmd_Reset) OTU(OCmd_Reset) ,XIC(Inp_Reset) ]CLR(Wrk_Sts);
   // If the Latch Defeat Input is ON (say, motor not running) and the stored interlock
   // status is clear (typically, after we get a reset in the rung above),
   // switch to "not latching" for all interlock inputs (regardless of Cfg_Latched).
   // This has the effect of keeping the Latch Enable work bit ON until a Reset is received.
   // Hence this is part of the "reset command processing" logic....
   3: EQU(Wrk_Sts,0)XIC(Inp_LatchDefeat)OTU(Wrk_LatchEnable);
   // ============================================================
   // INTERLOCK PROCESSING
   // ============================================================
   // This rung clears any bits in the stored Interlock status for which the
   // Input bit is OFF and the bit is NOT configured as Latched.
   // If the LatchDefeat input in OFF, set the internal Latch Enable work bit.
   // If this bit is ON, don't clear any latched bits with this rung (keep them latched).
   // If this bit is OFF, clear any bits that are NOT on in the input, whether
   // configured for latching or not!
   4: [XIO(Inp_LatchDefeat) OTL(Wrk_LatchEnable) ,XIC(Wrk_LatchEnable) OR(Cfg_Latched,Wrk_InpInv,Wrk_Intlk) ,XIO(Wrk_LatchEnable) MOV(Wrk_InpInv,Wrk_Intlk) ]AND(Wrk_Sts,Wrk_Intlk,Wrk_Sts);
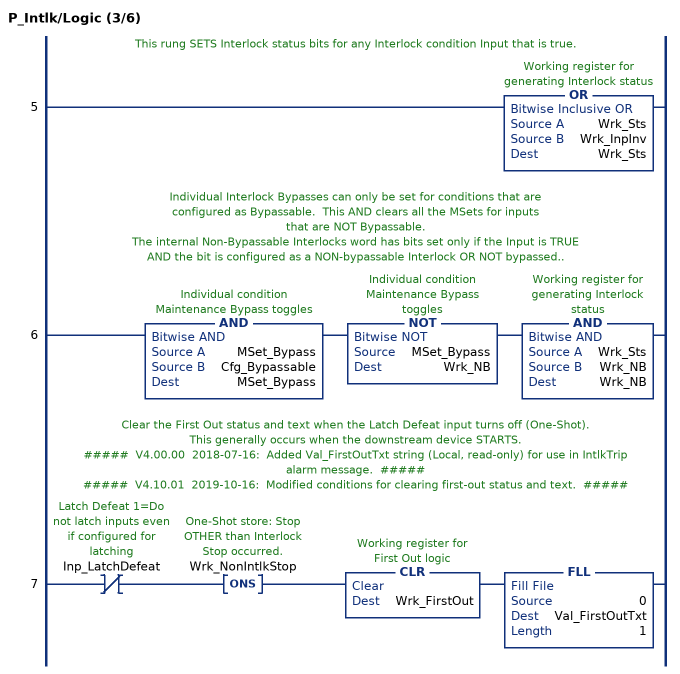
   // This rung SETS Interlock status bits for any Interlock condition Input that is true.
   5: OR(Wrk_Sts,Wrk_InpInv,Wrk_Sts);
   // Individual Interlock Bypasses can only be set for conditions that are
   // configured as Bypassable.  This AND clears all the MSets for inputs
   // that are NOT Bypassable.
   // The internal Non-Bypassable Interlocks word has bits set only if the Input is TRUE
   // AND the bit is configured as a NON-bypassable Interlock OR NOT bypassed..
   6: AND(MSet_Bypass,Cfg_Bypassable,MSet_Bypass)NOT(MSet_Bypass,Wrk_NB)AND(Wrk_Sts,Wrk_NB,Wrk_NB);
   // Clear the First Out status and text when the Latch Defeat input turns off (One-Shot).
   // This generally occurs when the downstream device STARTS.
   // #####  V4.00.00  2018-07-16:  Added Val_FirstOutTxt string (Local, read-only) for use in IntlkTrip alarm message.  #####
   // #####  V4.10.01  2019-10-16:  Modified conditions for clearing first-out status and text.  #####
   7: XIO(Inp_LatchDefeat)ONS(Wrk_NonIntlkStop)CLR(Wrk_FirstOut)FLL(0,Val_FirstOutTxt,1);
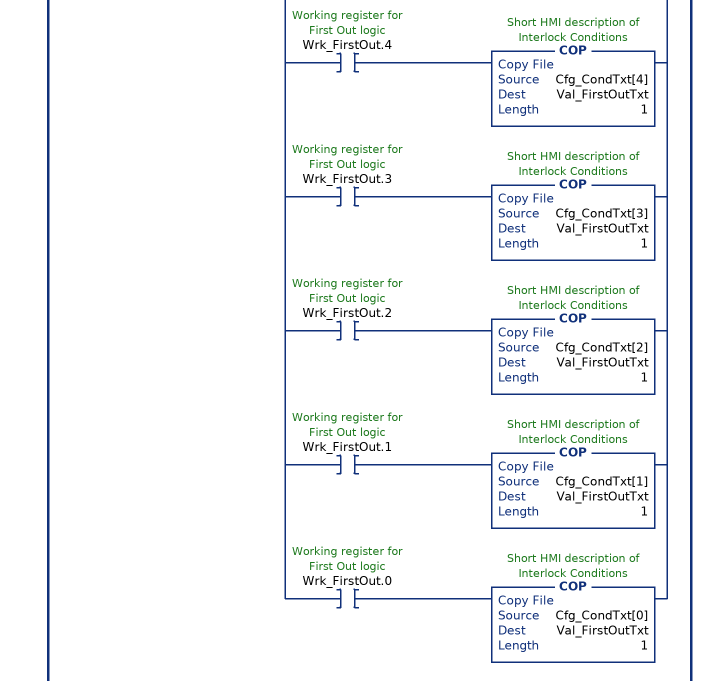
   // If an interlock condition occurs (which interlocks depends on the
   // bypass status!) and the Latch Defeat input is NOT set,
   // the equipment is running and will be shut down.
   // If this happens, record the First Out status.
   // #####  V4.00.00  2018-07-16:  Added Val_FirstOutTxt string (Local, read-only) for use in IntlkTrip alarm message.  #####
   // #####  V4.10.00  2019-03-08:  Changed type of Val_FirstOutTxt to STRING_Cond.  #####
   8: [XIO(Inp_BypActive) NEQ(Wrk_Sts,0) ,XIC(Inp_BypActive) NEQ(Wrk_NB,0) ]XIO(Inp_LatchDefeat)ONS(Wrk_SetFirstOut)[XIO(Inp_BypActive) CPT(Wrk_FirstOut,(Wrk_Sts)AND(NOT(Wrk_PrevSts))) ,XIC(Inp_BypActive) CPT(Wrk_FirstOut,(Wrk_NB)AND(NOT(Wrk_PrevSts))) ,NEQ(Wrk_FirstOut,0) [XIC(Wrk_FirstOut.15) COP(Cfg_CondTxt[15],Val_FirstOutTxt,1) ,XIC(Wrk_FirstOut.14) COP(Cfg_CondTxt[14],Val_FirstOutTxt,1) ,XIC(Wrk_FirstOut.13) COP(Cfg_CondTxt[13],Val_FirstOutTxt,1) ,XIC(Wrk_FirstOut.12) COP(Cfg_CondTxt[12],Val_FirstOutTxt,1) ,XIC(Wrk_FirstOut.11) COP(Cfg_CondTxt[11],Val_FirstOutTxt,1) ,XIC(Wrk_FirstOut.10) COP(Cfg_CondTxt[10],Val_FirstOutTxt,1) ,XIC(Wrk_FirstOut.9) COP(Cfg_CondTxt[9],Val_FirstOutTxt,1) ,XIC(Wrk_FirstOut.8) COP(Cfg_CondTxt[8],Val_FirstOutTxt,1) ,XIC(Wrk_FirstOut.7) COP(Cfg_CondTxt[7],Val_FirstOutTxt,1) ,XIC(Wrk_FirstOut.6) COP(Cfg_CondTxt[6],Val_FirstOutTxt,1) ,XIC(Wrk_FirstOut.5) COP(Cfg_CondTxt[5],Val_FirstOutTxt,1) ,XIC(Wrk_FirstOut.4) COP(Cfg_CondTxt[4],Val_FirstOutTxt,1) ,XIC(Wrk_FirstOut.3) COP(Cfg_CondTxt[3],Val_FirstOutTxt,1) ,XIC(Wrk_FirstOut.2) COP(Cfg_CondTxt[2],Val_FirstOutTxt,1) ,XIC(Wrk_FirstOut.1) COP(Cfg_CondTxt[1],Val_FirstOutTxt,1) ,XIC(Wrk_FirstOut.0) COP(Cfg_CondTxt[0],Val_FirstOutTxt,1) ] ];
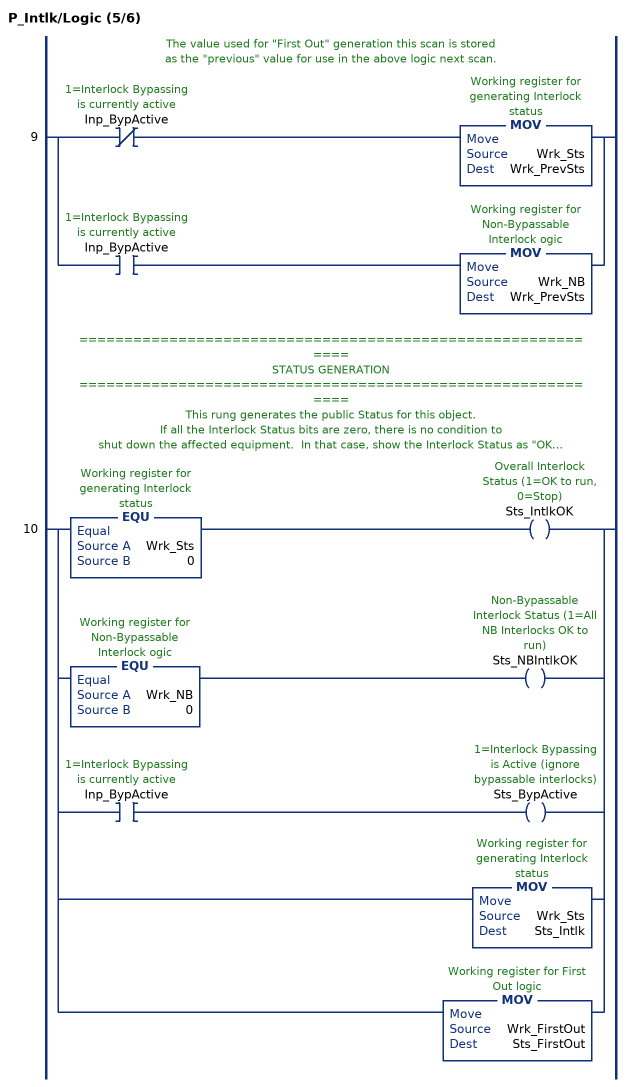
   // The value used for "First Out" generation this scan is stored
   // as the "previous" value for use in the above logic next scan.
   9: [XIO(Inp_BypActive) MOV(Wrk_Sts,Wrk_PrevSts) ,XIC(Inp_BypActive) MOV(Wrk_NB,Wrk_PrevSts) ];
   // ============================================================
   // STATUS GENERATION
   // ============================================================
   // This rung generates the public Status for this object.
   // If all the Interlock Status bits are zero, there is no condition to
   // shut down the affected equipment.  In that case, show the Interlock Status as "OK"
   // Similar logic applies for the Non-Bypassable Interlocks OK Status.
   // Also show the individual Interlock Status bits and the First Out Status bits.
   // NOTE:  Working registers are used to prevent outside writes to the Sts_xxx
   // parameters from affecting the state of this object!
   10: [[EQU(Wrk_Sts,0) OTE(Sts_IntlkOK) ,EQU(Wrk_NB,0) OTE(Sts_NBIntlkOK) ] ,XIC(Inp_BypActive) OTE(Sts_BypActive) ,MOV(Wrk_Sts,Sts_Intlk) ,MOV(Wrk_FirstOut,Sts_FirstOut) ];
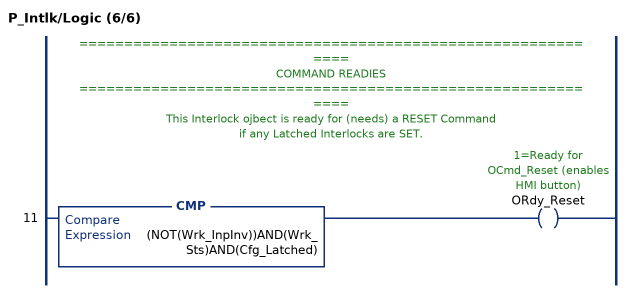
   // ============================================================
   // COMMAND READIES
   // ============================================================
   // This Interlock ojbect is ready for (needs) a RESET Command
   // if any Latched Interlocks are SET.
   11: CMP((NOT(Wrk_InpInv))AND(Wrk_Sts)AND(Cfg_Latched))OTE(ORdy_Reset);
END_ROUTINE
